FUNCTION_BLOCK EL1034
VAR
	_io : EL1xx4_Data;
	{attribute addProperty Name "WcState"}
	_wcState : WcStateInputToggle;
	{attribute addProperty Name "Info data"}
	_infoData : InfoDataBase;
END_VAR

PROPERTY IO : REFERENCE TO EL1xx4_Data
GET
IO REF= _io;
END_GET
END_PROPERTY

PROPERTY WcState : REFERENCE TO WcStateInputToggle
GET
WcState REF= _wcState;
END_GET
END_PROPERTY

END_FUNCTION_BLOCK

(* stored: Version 1.1.0.1, ProductVersion 3.1.4024.9
   POU EL1034: Id {9d24bd94-a141-0dd4-1cd0-5b2bc00129be}, SpecialFunc None
   Property IO: Id {1d026687-1bfa-0c6e-0df0-44f0b8fc55c1}
   Get Get: Id {23633b88-5815-0b4d-2091-d123a067f317}
   Property WcState: Id {b986f7cc-cee1-020d-116d-5f55a87cb0be}
   Get Get: Id {29a2f6c5-5874-0067-3111-0374f5c899ff} *)
